{attribute addProperty BoxType "ELX3152-0000-0016"}
{attribute addProperty Id "AI_Standard_ChannelAT %I*ARRAY[0..1] OF AI_Standard_Channel_087F71C76480WcStateAT %I*WcState_98A4DF7520.250InfoDataAT %I*InfoData_BC63D37F80100"}
{attribute addProperty CRC "4088362731"}
{attribute addProperty SizeInBites "146"}
{attribute addProperty SizeInBytes "18.25"}
TYPE ELX3152_C6F348DD :
STRUCT
	{attribute addProperty Name "AI_Standard_Channel"}
	AI_Standard_Channel : ARRAY[0..1] OF AI_Standard_Channel_087F71C7;
	{attribute addProperty Name "WcState"}
	WcState : WcState_98A4DF75;
	{attribute addProperty Name "InfoData"}
	InfoData : InfoData_BC63D37F;
END_STRUCT
END_TYPE

(* stored: Version 1.2.0.0, ProductVersion 3.1.4024.9
   DUT ELX3152_C6F348DD: Id {8c9adbd1-0c35-4296-8dda-4d038f3e1c5b} *)
